Yaskawa INFORM job: miniTRJ2.JBI

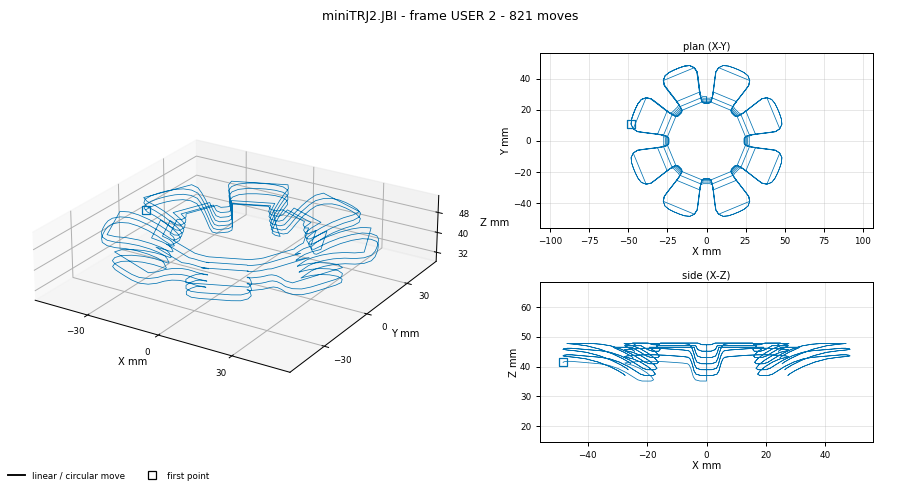
[picture p0: tool path of miniTRJ2.JBI in frame USER 2, 821 of 821 moves have a stored position in this frame; points joined in program order, loops and branches not executed]
/JOB
//NAME miniTRJ2
//POS
///NPOS 821,0,0,0,0,0
///USER 2
///TOOL 1
///POSTYPE USER
///RECTAN
///RCONF 1,0,0,0,0,0,0,0,0,0,0,0,0,0,0,0,0,0,0,0,0,0,0,0
C00000=-48.294,10.888,41.429,-176.7397,37.5709,0.0000
C00001=-47.960,14.116,41.642,-174.0482,36.6015,0.0000
C00002=-46.852,17.458,41.781,-171.5367,35.2544,0.0000
C00003=-45.474,20.785,41.781,148.5946,18.8544,0.0000
C00004=-43.894,23.932,41.642,148.9631,21.2691,0.0000
C00005=-41.848,26.450,41.429,149.6667,23.5333,0.0000
C00006=-38.982,27.526,41.216,150.5545,25.2242,0.0000
C00007=-35.890,26.937,40.953,151.2616,26.0383,0.0000
C00008=-32.968,24.818,40.447,151.5930,26.0678,0.0000
C00009=-29.853,22.391,39.399,151.8878,26.0592,0.0000
C00010=-27.005,20.165,37.988,152.1228,26.0805,0.0000
C00011=-24.775,18.500,36.587,152.2942,26.1489,0.0000
C00012=-23.134,17.826,35.561,152.5223,26.3895,0.0000
C00013=-21.719,18.610,35.152,153.0306,27.0004,0.0000
C00014=-20.847,19.522,35.134,152.8372,26.8332,0.0000
C00015=-20.193,20.193,35.146,151.5689,25.4617,0.0000
C00016=-19.522,20.846,35.134,150.3783,24.0388,0.0000
C00017=-18.610,21.719,35.152,150.2435,23.8342,0.0000
C00018=-17.826,23.134,35.561,150.7835,24.4140,0.0000
C00019=-18.500,24.775,36.587,150.9905,24.6675,0.0000
C00020=-20.165,27.005,37.988,151.0256,24.8329,0.0000
C00021=-22.391,29.853,39.399,150.9956,25.0433,0.0000
C00022=-24.818,32.968,40.447,150.9190,25.2991,0.0000
C00023=-26.937,35.890,40.953,150.8741,25.5955,0.0000
C00024=-27.526,38.982,41.216,151.5887,26.4057,0.0000
C00025=-26.450,41.848,41.429,153.2256,27.5826,0.0000
C00026=-23.932,43.894,41.642,155.5676,28.7163,0.0000
C00027=-20.785,45.474,41.781,158.1935,29.5466,0.0000
C00028=-17.458,46.852,41.781,144.4493,-6.9027,0.0000
C00029=-14.116,47.960,41.642,143.2501,-4.7750,0.0000
C00030=-10.888,48.294,41.429,142.3842,-2.5836,0.0000
C00031=-8.101,47.028,41.216,141.9857,-0.7523,0.0000
C00032=-6.331,44.425,40.953,141.9838,0.2816,0.0000
C00033=-5.763,40.861,40.447,142.1989,0.4896,0.0000
C00034=-5.276,36.942,39.399,142.4114,0.6478,0.0000
C00035=-4.837,33.354,37.988,142.5630,0.7963,0.0000
C00036=-4.437,30.601,36.587,142.6403,0.9460,0.0000
C00037=-3.753,28.963,35.561,142.6489,1.2616,0.0000
C00038=-2.199,28.517,35.152,142.6175,2.0220,0.0000
C00039=-0.937,28.545,35.134,142.5890,1.7848,0.0000
C00040=0.000,28.557,35.146,142.5588,-0.0019,0.0000
C00041=0.000,27.418,37.029,142.9317,-0.0022,0.0000
C00042=0.833,27.409,37.016,142.9601,-1.7182,0.0000
C00043=2.024,27.393,37.035,142.9884,-2.0087,0.0000
C00044=3.544,27.900,37.475,143.0157,-1.2641,0.0000
C00045=4.196,29.693,38.576,142.9980,-0.9669,0.0000
C00046=4.590,32.667,40.064,142.9030,-0.8249,0.0000
C00047=5.044,36.489,41.539,142.7233,-0.6720,0.0000
C00048=5.547,40.603,42.621,142.4757,-0.5065,0.0000
C00049=6.113,44.307,43.139,142.2242,-0.2970,0.0000
C00050=7.904,47.004,43.407,142.2019,0.7764,0.0000
C00051=10.737,48.321,43.623,142.6086,2.6858,0.0000
C00052=14.024,47.990,43.840,143.5265,4.9622,0.0000
C00053=17.428,46.864,43.981,144.8035,7.1518,0.0000
C00054=20.814,45.461,43.981,158.6858,-29.5002,0.0000
C00055=24.018,43.851,43.840,155.9451,-28.6807,0.0000
C00056=26.576,41.761,43.623,153.4943,-27.5200,0.0000
C00057=27.648,38.826,43.407,151.7943,-26.2899,0.0000
C00058=27.007,35.652,43.139,151.0729,-25.4348,0.0000
C00059=24.788,32.633,42.621,151.1478,-25.1145,0.0000
C00060=22.235,29.369,41.539,151.2491,-24.8312,0.0000
C00061=19.854,26.344,40.064,151.2998,-24.5999,0.0000
C00062=18.029,23.963,38.576,151.2850,-24.4296,0.0000
C00063=17.223,22.234,37.475,151.0981,-24.1854,0.0000
C00064=17.939,20.801,37.035,150.5715,-23.6167,0.0000
C00065=18.793,19.970,37.016,150.7430,-23.8628,0.0000
C00066=19.387,19.387,37.029,151.8889,-25.2262,0.0000
C00067=19.970,18.793,37.016,153.1137,-26.5489,0.0000
C00068=20.801,17.939,37.035,153.3424,-26.7551,0.0000
C00069=22.234,17.223,37.475,152.8415,-26.1602,0.0000
C00070=23.963,18.029,38.576,152.6183,-25.9402,0.0000
C00071=26.344,19.854,40.064,152.4370,-25.8893,0.0000
C00072=29.369,22.235,41.539,152.1749,-25.8826,0.0000
C00073=32.633,24.788,42.621,151.8451,-25.9079,0.0000
C00074=35.652,27.007,43.139,151.4812,-25.9004,0.0000
C00075=38.826,27.648,43.407,150.7258,-25.0713,0.0000
C00076=41.761,26.576,43.623,149.7917,-23.3150,0.0000
C00077=43.851,24.018,43.840,149.0753,-20.9529,0.0000
C00078=45.461,20.814,43.981,148.7289,-18.4429,0.0000
C00079=46.864,17.428,43.981,-171.2706,-34.8827,0.0000
C00080=47.990,14.024,43.840,-173.8375,-36.3149,0.0000
C00081=48.321,10.737,43.623,-176.6210,-37.3433,0.0000
C00082=47.004,7.904,43.407,-179.0175,-37.7940,0.0000
C00083=44.307,6.113,43.139,179.6243,-37.7752,0.0000
C00084=40.603,5.547,42.621,179.3613,-37.5226,0.0000
C00085=36.489,5.044,41.539,179.1555,-37.2737,0.0000
C00086=32.667,4.590,40.064,178.9658,-37.0926,0.0000
C00087=29.693,4.196,38.576,178.7894,-36.9959,0.0000
C00088=27.900,3.544,37.475,178.4177,-36.9738,0.0000
C00089=27.393,2.024,37.035,177.4851,-36.9851,0.0000
C00090=27.409,0.833,37.016,177.8479,-37.0204,0.0000
C00091=27.418,0.000,37.029,179.9973,-37.0683,0.0000
C00092=27.409,-0.832,37.016,-177.8467,-37.0204,0.0000
C00093=27.393,-2.024,37.035,-177.4859,-36.9851,0.0000
C00094=27.900,-3.544,37.475,-178.4183,-36.9738,0.0000
C00095=29.693,-4.196,38.576,-178.7900,-36.9959,0.0000
C00096=32.667,-4.590,40.064,-178.9664,-37.0925,0.0000
C00097=36.489,-5.044,41.539,-179.1560,-37.2737,0.0000
C00098=40.603,-5.547,42.621,-179.3619,-37.5226,0.0000
C00099=44.307,-6.113,43.139,-179.6249,-37.7752,0.0000
C00100=47.004,-7.904,43.407,179.0170,-37.7939,0.0000
C00101=48.321,-10.737,43.623,176.6207,-37.3433,0.0000
C00102=47.990,-14.024,43.840,173.8374,-36.3149,0.0000
C00103=46.864,-17.428,43.981,171.2706,-34.8827,0.0000
C00104=45.461,-20.814,43.981,-148.7290,-18.4429,0.0000
C00105=43.851,-24.018,43.840,-149.0753,-20.9529,0.0000
C00106=41.761,-26.576,43.623,-149.7918,-23.3152,0.0000
C00107=38.826,-27.648,43.407,-150.7260,-25.0716,0.0000
C00108=35.652,-27.007,43.139,-151.4815,-25.9008,0.0000
C00109=32.633,-24.788,42.621,-151.8454,-25.9083,0.0000
C00110=29.369,-22.235,41.539,-152.1752,-25.8829,0.0000
C00111=26.344,-19.854,40.064,-152.4373,-25.8897,0.0000
C00112=23.963,-18.029,38.576,-152.6186,-25.9406,0.0000
C00113=22.234,-17.223,37.475,-152.8418,-26.1606,0.0000
C00114=20.801,-17.939,37.035,-153.3429,-26.7556,0.0000
C00115=19.970,-18.793,37.016,-153.1131,-26.5482,0.0000
C00116=19.387,-19.387,37.029,-151.8919,-25.2296,0.0000
C00117=18.793,-19.970,37.016,-150.7424,-23.8621,0.0000
C00118=17.939,-20.801,37.035,-150.5720,-23.6172,0.0000
C00119=17.223,-22.234,37.475,-151.0984,-24.1858,0.0000
C00120=18.029,-23.963,38.576,-151.2853,-24.4300,0.0000
C00121=19.854,-26.344,40.064,-151.3001,-24.6002,0.0000
C00122=22.235,-29.369,41.539,-151.2494,-24.8316,0.0000
C00123=24.788,-32.633,42.621,-151.1482,-25.1149,0.0000
C00124=27.007,-35.652,43.139,-151.0733,-25.4352,0.0000
C00125=27.648,-38.826,43.407,-151.7946,-26.2902,0.0000
C00126=26.576,-41.761,43.623,-153.4945,-27.5201,0.0000
C00127=24.018,-43.851,43.840,-155.9452,-28.6808,0.0000
C00128=20.814,-45.461,43.981,-158.6857,-29.5002,0.0000
C00129=17.428,-46.864,43.981,-144.8035,7.1518,0.0000
C00130=14.024,-47.990,43.840,-143.5265,4.9622,0.0000
C00131=10.737,-48.321,43.623,-142.6086,2.6858,0.0000
C00132=7.904,-47.004,43.407,-142.2019,0.7764,0.0000
C00133=6.113,-44.307,43.139,-142.2242,-0.2970,0.0000
C00134=5.547,-40.603,42.621,-142.4757,-0.5065,0.0000
C00135=5.044,-36.489,41.539,-142.7233,-0.6720,0.0000
C00136=4.590,-32.667,40.064,-142.9030,-0.8249,0.0000
C00137=4.196,-29.693,38.576,-142.9980,-0.9669,0.0000
C00138=3.544,-27.900,37.475,-143.0157,-1.2641,0.0000
C00139=2.024,-27.393,37.035,-142.9884,-2.0087,0.0000
C00140=0.833,-27.409,37.016,-142.9601,-1.7182,0.0000
C00141=0.000,-27.418,37.029,-142.9317,-0.0022,0.0000
C00142=0.000,-27.418,37.029,-142.9317,-0.0022,0.0000
C00143=-0.832,-27.409,37.016,-142.9601,1.7191,0.0000
C00144=-2.024,-27.393,37.035,-142.9884,2.0080,0.0000
C00145=-3.544,-27.900,37.475,-143.0157,1.2636,0.0000
C00146=-4.196,-29.693,38.576,-142.9980,0.9664,0.0000
C00147=-4.590,-32.667,40.064,-142.9030,0.8245,0.0000
C00148=-5.044,-36.489,41.539,-142.7233,0.6716,0.0000
C00149=-5.547,-40.603,42.621,-142.4757,0.5061,0.0000
C00150=-6.113,-44.307,43.139,-142.2242,0.2965,0.0000
C00151=-7.904,-47.004,43.407,-142.2020,-0.7768,0.0000
C00152=-10.737,-48.321,43.623,-142.6086,-2.6860,0.0000
C00153=-14.024,-47.990,43.840,-143.5265,-4.9623,0.0000
C00154=-17.428,-46.864,43.981,-144.8035,-7.1518,0.0000
C00155=-20.814,-45.461,43.981,-158.6858,29.5002,0.0000
C00156=-24.018,-43.851,43.840,-155.9451,28.6807,0.0000
C00157=-26.576,-41.761,43.623,-153.4943,27.5200,0.0000
C00158=-27.648,-38.826,43.407,-151.7943,26.2899,0.0000
C00159=-27.007,-35.652,43.139,-151.0729,25.4348,0.0000
C00160=-24.788,-32.633,42.621,-151.1478,25.1145,0.0000
C00161=-22.235,-29.369,41.539,-151.2491,24.8312,0.0000
C00162=-19.854,-26.344,40.064,-151.2998,24.5999,0.0000
C00163=-18.029,-23.963,38.576,-151.2850,24.4296,0.0000
C00164=-17.223,-22.234,37.475,-151.0981,24.1854,0.0000
C00165=-17.939,-20.801,37.035,-150.5715,23.6167,0.0000
C00166=-18.793,-19.970,37.016,-150.7430,23.8628,0.0000
C00167=-19.387,-19.387,37.029,-151.8889,25.2262,0.0000
C00168=-19.970,-18.793,37.016,-153.1137,26.5489,0.0000
C00169=-20.801,-17.939,37.035,-153.3424,26.7551,0.0000
C00170=-22.234,-17.223,37.475,-152.8415,26.1602,0.0000
C00171=-23.963,-18.029,38.576,-152.6183,25.9402,0.0000
C00172=-26.344,-19.854,40.064,-152.4370,25.8893,0.0000
C00173=-29.369,-22.235,41.539,-152.1749,25.8826,0.0000
C00174=-32.633,-24.788,42.621,-151.8451,25.9079,0.0000
C00175=-35.652,-27.007,43.139,-151.4812,25.9004,0.0000
C00176=-38.826,-27.648,43.407,-150.7258,25.0713,0.0000
C00177=-41.761,-26.576,43.623,-149.7917,23.3150,0.0000
C00178=-43.851,-24.018,43.840,-149.0753,20.9529,0.0000
C00179=-45.461,-20.814,43.981,-148.7289,18.4429,0.0000
C00180=-46.864,-17.428,43.981,171.2706,34.8827,0.0000
C00181=-47.990,-14.024,43.840,173.8375,36.3149,0.0000
C00182=-48.321,-10.737,43.623,176.6210,37.3433,0.0000
C00183=-47.004,-7.904,43.407,179.0175,37.7940,0.0000
C00184=-44.307,-6.113,43.139,-179.6243,37.7752,0.0000
C00185=-40.603,-5.547,42.621,-179.3613,37.5226,0.0000
C00186=-36.489,-5.044,41.539,-179.1555,37.2737,0.0000
C00187=-32.667,-4.590,40.064,-178.9658,37.0926,0.0000
C00188=-29.693,-4.196,38.576,-178.7894,36.9959,0.0000
C00189=-27.900,-3.544,37.475,-178.4177,36.9738,0.0000
C00190=-27.393,-2.024,37.035,-177.4851,36.9851,0.0000
C00191=-27.409,-0.833,37.016,-177.8479,37.0204,0.0000
C00192=-27.418,0.000,37.029,-179.9973,37.0683,0.0000
C00193=-27.409,0.832,37.016,177.8467,37.0204,0.0000
C00194=-27.393,2.024,37.035,177.4859,36.9851,0.0000
C00195=-27.900,3.544,37.475,178.4183,36.9738,0.0000
C00196=-29.693,4.196,38.576,178.7900,36.9959,0.0000
C00197=-32.667,4.590,40.064,178.9664,37.0925,0.0000
C00198=-36.489,5.044,41.539,179.1560,37.2737,0.0000
C00199=-40.603,5.547,42.621,179.3619,37.5226,0.0000
C00200=-44.307,6.113,43.139,179.6249,37.7752,0.0000
C00201=-47.004,7.904,43.407,-179.0170,37.7939,0.0000
C00202=-48.321,10.737,43.623,-176.6207,37.3433,0.0000
C00203=-47.990,14.024,43.840,-173.8374,36.3149,0.0000
C00204=-46.864,17.428,43.981,-171.2706,34.8827,0.0000
C00205=-45.461,20.814,43.981,148.7290,18.4429,0.0000
C00206=-43.851,24.018,43.840,149.0753,20.9529,0.0000
C00207=-41.761,26.576,43.623,149.7918,23.3152,0.0000
C00208=-38.826,27.648,43.407,150.7260,25.0716,0.0000
C00209=-35.652,27.007,43.139,151.4815,25.9008,0.0000
C00210=-32.633,24.788,42.621,151.8454,25.9083,0.0000
C00211=-29.369,22.235,41.539,152.1752,25.8829,0.0000
C00212=-26.344,19.854,40.064,152.4373,25.8897,0.0000
C00213=-23.963,18.029,38.576,152.6186,25.9406,0.0000
C00214=-22.234,17.223,37.475,152.8418,26.1606,0.0000
C00215=-20.801,17.939,37.035,153.3429,26.7556,0.0000
C00216=-19.970,18.793,37.016,153.1131,26.5482,0.0000
C00217=-19.387,19.387,37.029,151.8919,25.2296,0.0000
C00218=-18.793,19.970,37.016,150.7424,23.8621,0.0000
C00219=-17.939,20.801,37.035,150.5720,23.6172,0.0000
C00220=-17.223,22.234,37.475,151.0984,24.1858,0.0000
C00221=-18.029,23.963,38.576,151.2853,24.4300,0.0000
C00222=-19.854,26.344,40.064,151.3001,24.6002,0.0000
C00223=-22.235,29.369,41.539,151.2494,24.8316,0.0000
C00224=-24.788,32.633,42.621,151.1482,25.1149,0.0000
C00225=-27.007,35.652,43.139,151.0733,25.4352,0.0000
C00226=-27.648,38.826,43.407,151.7946,26.2902,0.0000
C00227=-26.576,41.761,43.623,153.4945,27.5201,0.0000
C00228=-24.018,43.851,43.840,155.9452,28.6808,0.0000
C00229=-20.814,45.461,43.981,158.6857,29.5002,0.0000
C00230=-17.428,46.864,43.981,144.8035,-7.1518,0.0000
C00231=-14.024,47.990,43.840,143.5265,-4.9623,0.0000
C00232=-10.737,48.321,43.623,142.6086,-2.6860,0.0000
C00233=-7.904,47.004,43.407,142.2020,-0.7768,0.0000
C00234=-6.113,44.307,43.139,142.2242,0.2965,0.0000
C00235=-5.547,40.603,42.621,142.4757,0.5061,0.0000
C00236=-5.044,36.489,41.539,142.7233,0.6716,0.0000
C00237=-4.590,32.667,40.064,142.9030,0.8245,0.0000
C00238=-4.196,29.693,38.576,142.9980,0.9664,0.0000
C00239=-3.544,27.900,37.475,143.0157,1.2636,0.0000
C00240=-2.024,27.393,37.035,142.9884,2.0080,0.0000
C00241=-0.832,27.409,37.016,142.9601,1.7191,0.0000
C00242=0.000,27.418,37.029,142.9317,-0.0022,0.0000
C00243=0.000,26.383,38.970,143.3333,-0.0024,0.0000
C00244=0.738,26.377,38.956,143.3599,-1.6506,0.0000
C00245=1.865,26.371,38.977,143.3880,-1.9910,0.0000
C00246=3.355,26.945,39.448,143.4111,-1.2604,0.0000
C00247=3.987,28.902,40.618,143.3831,-0.9770,0.0000
C00248=4.387,32.102,42.180,143.2683,-0.8359,0.0000
C00249=4.868,36.145,43.705,143.0598,-0.6708,0.0000
C00250=5.395,40.422,44.808,142.7788,-0.4897,0.0000
C00251=5.967,44.227,45.333,142.4944,-0.2702,0.0000
C00252=7.777,46.989,45.603,142.4530,0.8448,0.0000
C00253=10.643,48.338,45.821,142.8730,2.8264,0.0000
C00254=13.968,48.009,46.039,143.8450,5.1732,0.0000
C00255=17.410,46.871,46.181,145.1966,7.4059,0.0000
C00256=20.832,45.453,46.181,159.2143,-29.4305,0.0000
C00257=24.070,43.824,46.039,156.3761,-28.6352,0.0000
C00258=26.655,41.706,45.821,153.8250,-27.4611,0.0000
C00259=27.727,38.725,45.603,152.0606,-26.1867,0.0000
C00260=27.054,35.493,45.333,151.3259,-25.2884,0.0000
C00261=24.768,32.397,44.808,151.4217,-24.9398,0.0000
C00262=22.116,29.001,43.705,151.5403,-24.6233,0.0000
C00263=19.598,25.801,42.180,151.6069,-24.3643,0.0000
C00264=17.618,23.256,40.618,151.6092,-24.1825,0.0000
C00265=16.680,21.426,39.448,151.4402,-23.9431,0.0000
C00266=17.329,19.966,38.977,150.9260,-23.3840,0.0000
C00267=18.130,19.173,38.956,151.1318,-23.6688,0.0000
C00268=18.656,18.656,38.970,152.2350,-24.9751,0.0000
C00269=19.173,18.130,38.956,153.4120,-26.2443,0.0000
C00270=19.966,17.329,38.977,153.6756,-26.4885,0.0000
C00271=21.426,16.680,39.448,153.1805,-25.9082,0.0000
C00272=23.256,17.618,40.618,152.9579,-25.7059,0.0000
C00273=25.801,19.598,42.180,152.7605,-25.6685,0.0000
C00274=29.001,22.116,43.705,152.4654,-25.6709,0.0000
C00275=32.397,24.768,44.808,152.0964,-25.7056,0.0000
C00276=35.493,27.054,45.333,151.6977,-25.7114,0.0000
C00277=38.725,27.727,45.603,150.8971,-24.8625,0.0000
C00278=41.706,26.655,45.821,149.9252,-23.0422,0.0000
C00279=43.824,24.070,46.039,149.2067,-20.5923,0.0000
C00280=45.453,20.832,46.181,148.8912,-18.0037,0.0000
C00281=46.871,17.410,46.181,-171.0047,-34.4718,0.0000
C00282=48.009,13.968,46.039,-173.6022,-35.9847,0.0000
C00283=48.338,10.643,45.821,-176.4566,-37.0743,0.0000
C00284=46.989,7.777,45.603,-178.9345,-37.5422,0.0000
C00285=44.227,5.967,45.333,179.6594,-37.5052,0.0000
C00286=40.422,5.395,44.808,179.3850,-37.2196,0.0000
C00287=36.145,4.868,43.705,179.1607,-36.9373,0.0000
C00288=32.102,4.387,42.180,178.9570,-36.7271,0.0000
C00289=28.902,3.987,40.618,178.7829,-36.6107,0.0000
C00290=26.945,3.355,39.448,178.4304,-36.5786,0.0000
C00291=26.371,1.865,38.977,177.5201,-36.5863,0.0000
C00292=26.377,0.738,38.956,177.9433,-36.6224,0.0000
C00293=26.383,0.000,38.970,179.9970,-36.6667,0.0000
C00294=26.377,-0.738,38.956,-177.9417,-36.6224,0.0000
C00295=26.371,-1.865,38.977,-177.5209,-36.5863,0.0000
C00296=26.945,-3.355,39.448,-178.4310,-36.5786,0.0000
C00297=28.902,-3.987,40.618,-178.7834,-36.6107,0.0000
C00298=32.102,-4.387,42.180,-178.9576,-36.7271,0.0000
C00299=36.145,-4.868,43.705,-179.1613,-36.9372,0.0000
C00300=40.422,-5.395,44.808,-179.3856,-37.2196,0.0000
C00301=44.227,-5.967,45.333,-179.6600,-37.5051,0.0000
C00302=46.989,-7.777,45.603,178.9341,-37.5421,0.0000
C00303=48.338,-10.643,45.821,176.4564,-37.0742,0.0000
C00304=48.009,-13.968,46.039,173.6022,-35.9847,0.0000
C00305=46.871,-17.410,46.181,171.0047,-34.4718,0.0000
C00306=45.453,-20.832,46.181,-148.8912,-18.0037,0.0000
C00307=43.824,-24.070,46.039,-149.2068,-20.5924,0.0000
C00308=41.706,-26.655,45.821,-149.9253,-23.0424,0.0000
C00309=38.725,-27.727,45.603,-150.8973,-24.8628,0.0000
C00310=35.493,-27.054,45.333,-151.6980,-25.7118,0.0000
C00311=32.397,-24.768,44.808,-152.0967,-25.7060,0.0000
C00312=29.001,-22.116,43.705,-152.4657,-25.6713,0.0000
C00313=25.801,-19.598,42.180,-152.7608,-25.6688,0.0000
C00314=23.256,-17.618,40.618,-152.9582,-25.7062,0.0000
C00315=21.426,-16.680,39.448,-153.1809,-25.9086,0.0000
C00316=19.966,-17.329,38.977,-153.6761,-26.4890,0.0000
C00317=19.173,-18.130,38.956,-153.4112,-26.2433,0.0000
C00318=18.656,-18.656,38.970,-152.2384,-24.9789,0.0000
C00319=18.130,-19.173,38.956,-151.1310,-23.6679,0.0000
C00320=17.329,-19.966,38.977,-150.9265,-23.3846,0.0000
C00321=16.680,-21.426,39.448,-151.4406,-23.9435,0.0000
C00322=17.618,-23.256,40.618,-151.6095,-24.1829,0.0000
C00323=19.598,-25.801,42.180,-151.6072,-24.3646,0.0000
C00324=22.116,-29.001,43.705,-151.5406,-24.6236,0.0000
C00325=24.768,-32.397,44.808,-151.4221,-24.9401,0.0000
C00326=27.054,-35.493,45.333,-151.3263,-25.2888,0.0000
C00327=27.727,-38.725,45.603,-152.0609,-26.1870,0.0000
C00328=26.655,-41.706,45.821,-153.8251,-27.4613,0.0000
C00329=24.070,-43.824,46.039,-156.3762,-28.6353,0.0000
C00330=20.832,-45.453,46.181,-159.2143,-29.4305,0.0000
C00331=17.410,-46.871,46.181,-145.1966,7.4059,0.0000
C00332=13.968,-48.009,46.039,-143.8450,5.1732,0.0000
C00333=10.643,-48.338,45.821,-142.8730,2.8264,0.0000
C00334=7.777,-46.989,45.603,-142.4530,0.8448,0.0000
C00335=5.967,-44.227,45.333,-142.4944,-0.2702,0.0000
C00336=5.395,-40.422,44.808,-142.7788,-0.4897,0.0000
C00337=4.868,-36.145,43.705,-143.0598,-0.6708,0.0000
C00338=4.387,-32.102,42.180,-143.2683,-0.8359,0.0000
C00339=3.987,-28.902,40.618,-143.3831,-0.9770,0.0000
C00340=3.355,-26.945,39.448,-143.4111,-1.2604,0.0000
C00341=1.865,-26.371,38.977,-143.3880,-1.9910,0.0000
C00342=0.738,-26.377,38.956,-143.3599,-1.6506,0.0000
C00343=0.000,-26.383,38.970,-143.3333,-0.0024,0.0000
C00344=0.000,-26.383,38.970,-143.3333,-0.0024,0.0000
C00345=-0.738,-26.377,38.956,-143.3599,1.6518,0.0000
C00346=-1.865,-26.371,38.977,-143.3880,1.9904,0.0000
C00347=-3.355,-26.945,39.448,-143.4111,1.2599,0.0000
C00348=-3.987,-28.902,40.618,-143.3831,0.9765,0.0000
C00349=-4.387,-32.102,42.180,-143.2684,0.8355,0.0000
C00350=-4.868,-36.145,43.705,-143.0598,0.6703,0.0000
C00351=-5.395,-40.422,44.808,-142.7788,0.4893,0.0000
C00352=-5.967,-44.227,45.333,-142.4944,0.2697,0.0000
C00353=-7.777,-46.989,45.603,-142.4531,-0.8452,0.0000
C00354=-10.643,-48.338,45.821,-142.8730,-2.8266,0.0000
C00355=-13.968,-48.009,46.039,-143.8450,-5.1732,0.0000
C00356=-17.410,-46.871,46.181,-145.1966,-7.4059,0.0000
C00357=-20.832,-45.453,46.181,-159.2143,29.4305,0.0000
C00358=-24.070,-43.824,46.039,-156.3761,28.6352,0.0000
C00359=-26.655,-41.706,45.821,-153.8250,27.4611,0.0000
C00360=-27.727,-38.725,45.603,-152.0606,26.1867,0.0000
C00361=-27.054,-35.493,45.333,-151.3259,25.2884,0.0000
C00362=-24.768,-32.397,44.808,-151.4217,24.9398,0.0000
C00363=-22.116,-29.001,43.705,-151.5403,24.6233,0.0000
C00364=-19.598,-25.801,42.180,-151.6069,24.3643,0.0000
C00365=-17.618,-23.256,40.618,-151.6092,24.1825,0.0000
C00366=-16.680,-21.426,39.448,-151.4402,23.9431,0.0000
C00367=-17.329,-19.966,38.977,-150.9260,23.3840,0.0000
C00368=-18.130,-19.173,38.956,-151.1318,23.6688,0.0000
C00369=-18.656,-18.656,38.970,-152.2350,24.9751,0.0000
C00370=-19.173,-18.130,38.956,-153.4120,26.2443,0.0000
C00371=-19.966,-17.329,38.977,-153.6756,26.4885,0.0000
C00372=-21.426,-16.680,39.448,-153.1805,25.9082,0.0000
C00373=-23.256,-17.618,40.618,-152.9579,25.7059,0.0000
C00374=-25.801,-19.598,42.180,-152.7605,25.6685,0.0000
C00375=-29.001,-22.116,43.705,-152.4654,25.6709,0.0000
C00376=-32.397,-24.768,44.808,-152.0964,25.7056,0.0000
C00377=-35.493,-27.054,45.333,-151.6977,25.7114,0.0000
C00378=-38.725,-27.727,45.603,-150.8971,24.8625,0.0000
C00379=-41.706,-26.655,45.821,-149.9252,23.0422,0.0000
C00380=-43.824,-24.070,46.039,-149.2067,20.5923,0.0000
C00381=-45.453,-20.832,46.181,-148.8912,18.0037,0.0000
C00382=-46.871,-17.410,46.181,171.0047,34.4718,0.0000
C00383=-48.009,-13.968,46.039,173.6022,35.9847,0.0000
C00384=-48.338,-10.643,45.821,176.4566,37.0743,0.0000
C00385=-46.989,-7.777,45.603,178.9345,37.5422,0.0000
C00386=-44.227,-5.967,45.333,-179.6594,37.5052,0.0000
C00387=-40.422,-5.395,44.808,-179.3850,37.2196,0.0000
C00388=-36.145,-4.868,43.705,-179.1607,36.9373,0.0000
C00389=-32.102,-4.387,42.180,-178.9570,36.7271,0.0000
C00390=-28.902,-3.987,40.618,-178.7829,36.6107,0.0000
C00391=-26.945,-3.355,39.448,-178.4304,36.5786,0.0000
C00392=-26.371,-1.865,38.977,-177.5201,36.5863,0.0000
C00393=-26.377,-0.738,38.956,-177.9433,36.6224,0.0000
C00394=-26.383,0.000,38.970,-179.9970,36.6667,0.0000
C00395=-26.377,0.738,38.956,177.9417,36.6224,0.0000
C00396=-26.371,1.865,38.977,177.5209,36.5863,0.0000
C00397=-26.945,3.355,39.448,178.4310,36.5786,0.0000
C00398=-28.902,3.987,40.618,178.7834,36.6107,0.0000
C00399=-32.102,4.387,42.180,178.9576,36.7271,0.0000
C00400=-36.145,4.868,43.705,179.1613,36.9372,0.0000
C00401=-40.422,5.395,44.808,179.3856,37.2196,0.0000
C00402=-44.227,5.967,45.333,179.6600,37.5051,0.0000
C00403=-46.989,7.777,45.603,-178.9341,37.5421,0.0000
C00404=-48.338,10.643,45.821,-176.4564,37.0742,0.0000
C00405=-48.009,13.968,46.039,-173.6022,35.9847,0.0000
C00406=-46.871,17.410,46.181,-171.0047,34.4718,0.0000
C00407=-45.453,20.832,46.181,148.8912,18.0037,0.0000
C00408=-43.824,24.070,46.039,149.2068,20.5924,0.0000
C00409=-41.706,26.655,45.821,149.9253,23.0424,0.0000
C00410=-38.725,27.727,45.603,150.8973,24.8628,0.0000
C00411=-35.493,27.054,45.333,151.6980,25.7118,0.0000
C00412=-32.397,24.768,44.808,152.0967,25.7060,0.0000
C00413=-29.001,22.116,43.705,152.4657,25.6713,0.0000
C00414=-25.801,19.598,42.180,152.7608,25.6688,0.0000
C00415=-23.256,17.618,40.618,152.9582,25.7062,0.0000
C00416=-21.426,16.680,39.448,153.1809,25.9086,0.0000
C00417=-19.966,17.329,38.977,153.6761,26.4890,0.0000
C00418=-19.173,18.130,38.956,153.4112,26.2433,0.0000
C00419=-18.656,18.656,38.970,152.2384,24.9789,0.0000
C00420=-18.130,19.173,38.956,151.1310,23.6679,0.0000
C00421=-17.329,19.966,38.977,150.9265,23.3846,0.0000
C00422=-16.680,21.426,39.448,151.4406,23.9435,0.0000
C00423=-17.618,23.256,40.618,151.6095,24.1829,0.0000
C00424=-19.598,25.801,42.180,151.6072,24.3646,0.0000
C00425=-22.116,29.001,43.705,151.5406,24.6236,0.0000
C00426=-24.768,32.397,44.808,151.4221,24.9401,0.0000
C00427=-27.054,35.493,45.333,151.3263,25.2888,0.0000
C00428=-27.727,38.725,45.603,152.0609,26.1870,0.0000
C00429=-26.655,41.706,45.821,153.8251,27.4613,0.0000
C00430=-24.070,43.824,46.039,156.3762,28.6353,0.0000
C00431=-20.832,45.453,46.181,159.2143,29.4305,0.0000
C00432=-17.410,46.871,46.181,145.1966,-7.4059,0.0000
C00433=-13.968,48.009,46.039,143.8450,-5.1732,0.0000
C00434=-10.643,48.338,45.821,142.8730,-2.8266,0.0000
C00435=-7.777,46.989,45.603,142.4531,-0.8452,0.0000
C00436=-5.967,44.227,45.333,142.4944,0.2697,0.0000
C00437=-5.395,40.422,44.808,142.7788,0.4893,0.0000
C00438=-4.868,36.145,43.705,143.0598,0.6703,0.0000
C00439=-4.387,32.102,42.180,143.2684,0.8355,0.0000
C00440=-3.987,28.902,40.618,143.3831,0.9765,0.0000
C00441=-3.355,26.945,39.448,143.4111,1.2599,0.0000
C00442=-1.865,26.371,38.977,143.3880,1.9904,0.0000
C00443=-0.738,26.377,38.956,143.3599,1.6518,0.0000
C00444=0.000,26.383,38.970,143.3333,-0.0024,0.0000
C00445=0.000,25.483,40.978,143.7606,-0.0027,0.0000
C00446=0.656,25.479,40.963,143.7854,-1.5834,0.0000
C00447=1.726,25.483,40.985,143.8134,-1.9683,0.0000
C00448=3.194,26.129,41.485,143.8318,-1.2486,0.0000
C00449=3.816,28.261,42.716,143.7915,-0.9729,0.0000
C00450=4.237,31.687,44.335,143.6546,-0.8247,0.0000
C00451=4.757,35.929,45.891,143.4171,-0.6383,0.0000
C00452=5.317,40.329,47.005,143.1061,-0.4321,0.0000
C00453=5.904,44.193,47.531,142.7941,-0.1927,0.0000
C00454=7.727,46.983,47.803,142.7410,0.9664,0.0000
C00455=27.758,38.686,47.803,152.3956,-26.1014,0.0000
C00456=27.074,35.424,47.531,151.6387,-25.1629,0.0000
C00457=24.758,32.277,47.005,151.7437,-24.7813,0.0000
C00458=22.041,28.769,45.891,151.8698,-24.4263,0.0000
C00459=19.410,25.402,44.335,151.9459,-24.1324,0.0000
C00460=17.285,22.682,42.716,151.9617,-23.9312,0.0000
C00461=16.217,20.734,41.485,151.8082,-23.6905,0.0000
C00462=16.798,19.240,40.985,151.3046,-23.1385,0.0000
C00463=17.553,18.480,40.963,151.5411,-23.4575,0.0000
C00464=18.019,18.019,40.978,152.6017,-24.7072,0.0000
C00465=18.480,17.553,40.963,153.7314,-25.9231,0.0000
C00466=19.240,16.798,40.985,154.0260,-26.2010,0.0000
C00467=20.735,16.217,41.485,153.5342,-25.6332,0.0000
C00468=22.682,17.285,42.716,153.3064,-25.4451,0.0000
C00469=25.402,19.410,44.335,153.0852,-25.4166,0.0000
C00470=28.769,22.041,45.891,152.7509,-25.4213,0.0000
C00471=32.277,24.758,47.005,152.3396,-25.4559,0.0000
C00472=35.424,27.074,47.531,151.9041,-25.4640,0.0000
C00473=38.686,27.758,47.803,151.0634,-24.5889,0.0000
C00474=46.983,7.727,47.803,-178.7859,-37.2528,0.0000
C00475=44.193,5.904,47.531,179.7580,-37.2056,0.0000
C00476=40.329,5.317,47.005,179.4597,-36.8927,0.0000
C00477=35.929,4.757,45.891,179.2051,-36.5803,0.0000
C00478=31.687,4.237,44.335,178.9761,-36.3410,0.0000
C00479=28.261,3.816,42.716,178.7942,-36.2024,0.0000
C00480=26.129,3.194,41.485,178.4534,-36.1582,0.0000
C00481=25.483,1.726,40.985,177.5617,-36.1619,0.0000
C00482=25.479,0.656,40.963,178.0377,-36.1986,0.0000
C00483=25.483,0.000,40.978,179.9967,-36.2394,0.0000
C00484=25.479,-0.655,40.963,-178.0358,-36.1986,0.0000
C00485=25.483,-1.727,40.985,-177.5626,-36.1619,0.0000
C00486=26.129,-3.194,41.485,-178.4540,-36.1582,0.0000
C00487=28.261,-3.816,42.716,-178.7948,-36.2024,0.0000
C00488=31.687,-4.237,44.335,-178.9767,-36.3410,0.0000
C00489=35.929,-4.757,45.891,-179.2056,-36.5803,0.0000
C00490=40.329,-5.317,47.005,-179.4603,-36.8926,0.0000
C00491=44.193,-5.904,47.531,-179.7586,-37.2056,0.0000
C00492=46.983,-7.727,47.803,178.7854,-37.2528,0.0000
C00493=38.686,-27.758,47.803,-151.0636,-24.5892,0.0000
C00494=35.424,-27.074,47.531,-151.9044,-25.4644,0.0000
C00495=32.277,-24.758,47.005,-152.3399,-25.4563,0.0000
C00496=28.769,-22.041,45.891,-152.7512,-25.4217,0.0000
C00497=25.402,-19.410,44.335,-153.0855,-25.4169,0.0000
C00498=22.682,-17.285,42.716,-153.3067,-25.4455,0.0000
C00499=20.734,-16.217,41.485,-153.5345,-25.6335,0.0000
C00500=19.240,-16.798,40.985,-154.0265,-26.2015,0.0000
C00501=18.480,-17.553,40.963,-153.7302,-25.9220,0.0000
C00502=18.019,-18.019,40.978,-152.6054,-24.7113,0.0000
C00503=17.553,-18.480,40.963,-151.5400,-23.4562,0.0000
C00504=16.798,-19.240,40.985,-151.3050,-23.1390,0.0000
C00505=16.217,-20.735,41.485,-151.8085,-23.6909,0.0000
C00506=17.285,-22.682,42.716,-151.9620,-23.9315,0.0000
C00507=19.410,-25.402,44.335,-151.9462,-24.1327,0.0000
C00508=22.041,-28.769,45.891,-151.8701,-24.4266,0.0000
C00509=24.758,-32.277,47.005,-151.7440,-24.7817,0.0000
C00510=27.074,-35.424,47.531,-151.6391,-25.1632,0.0000
C00511=27.758,-38.686,47.803,-152.3959,-26.1016,0.0000
C00512=7.727,-46.983,47.803,-142.7410,0.9664,0.0000
C00513=5.904,-44.193,47.531,-142.7941,-0.1927,0.0000
C00514=5.317,-40.329,47.005,-143.1061,-0.4321,0.0000
C00515=4.757,-35.929,45.891,-143.4171,-0.6383,0.0000
C00516=4.237,-31.687,44.335,-143.6546,-0.8247,0.0000
C00517=3.816,-28.261,42.716,-143.7915,-0.9729,0.0000
C00518=3.194,-26.129,41.485,-143.8318,-1.2486,0.0000
C00519=1.726,-25.483,40.985,-143.8134,-1.9683,0.0000
C00520=0.656,-25.479,40.963,-143.7854,-1.5834,0.0000
C00521=0.000,-25.483,40.978,-143.7606,-0.0027,0.0000
C00522=0.000,-25.483,40.978,-143.7606,-0.0027,0.0000
C00523=-0.655,-25.479,40.963,-143.7854,1.5850,0.0000
C00524=-1.727,-25.483,40.985,-143.8134,1.9677,0.0000
C00525=-3.194,-26.129,41.485,-143.8318,1.2481,0.0000
C00526=-3.816,-28.261,42.716,-143.7915,0.9725,0.0000
C00527=-4.237,-31.687,44.335,-143.6547,0.8243,0.0000
C00528=-4.757,-35.929,45.891,-143.4171,0.6379,0.0000
C00529=-5.317,-40.329,47.005,-143.1061,0.4317,0.0000
C00530=-5.904,-44.193,47.531,-142.7942,0.1923,0.0000
C00531=-7.727,-46.983,47.803,-142.7410,-0.9667,0.0000
C00532=-27.758,-38.686,47.803,-152.3956,26.1014,0.0000
C00533=-27.074,-35.424,47.531,-151.6387,25.1629,0.0000
C00534=-24.758,-32.277,47.005,-151.7437,24.7813,0.0000
C00535=-22.041,-28.769,45.891,-151.8698,24.4263,0.0000
C00536=-19.410,-25.402,44.335,-151.9459,24.1324,0.0000
C00537=-17.285,-22.682,42.716,-151.9617,23.9312,0.0000
C00538=-16.217,-20.734,41.485,-151.8082,23.6905,0.0000
C00539=-16.798,-19.240,40.985,-151.3046,23.1385,0.0000
C00540=-17.553,-18.480,40.963,-151.5411,23.4575,0.0000
C00541=-18.019,-18.019,40.978,-152.6017,24.7072,0.0000
C00542=-18.480,-17.553,40.963,-153.7314,25.9231,0.0000
C00543=-19.240,-16.798,40.985,-154.0260,26.2010,0.0000
C00544=-20.735,-16.217,41.485,-153.5342,25.6332,0.0000
C00545=-22.682,-17.285,42.716,-153.3064,25.4451,0.0000
C00546=-25.402,-19.410,44.335,-153.0852,25.4166,0.0000
C00547=-28.769,-22.041,45.891,-152.7509,25.4213,0.0000
C00548=-32.277,-24.758,47.005,-152.3396,25.4559,0.0000
C00549=-35.424,-27.074,47.531,-151.9041,25.4640,0.0000
C00550=-38.686,-27.758,47.803,-151.0634,24.5889,0.0000
C00551=-46.983,-7.727,47.803,178.7859,37.2528,0.0000
C00552=-44.193,-5.904,47.531,-179.7580,37.2056,0.0000
C00553=-40.329,-5.317,47.005,-179.4597,36.8927,0.0000
C00554=-35.929,-4.757,45.891,-179.2051,36.5803,0.0000
C00555=-31.687,-4.237,44.335,-178.9761,36.3410,0.0000
C00556=-28.261,-3.816,42.716,-178.7942,36.2024,0.0000
C00557=-26.129,-3.194,41.485,-178.4534,36.1582,0.0000
C00558=-25.483,-1.726,40.985,-177.5617,36.1619,0.0000
C00559=-25.479,-0.656,40.963,-178.0377,36.1986,0.0000
C00560=-25.483,0.000,40.978,-179.9967,36.2394,0.0000
C00561=-25.479,0.655,40.963,178.0358,36.1986,0.0000
C00562=-25.483,1.727,40.985,177.5626,36.1619,0.0000
C00563=-26.129,3.194,41.485,178.4540,36.1582,0.0000
C00564=-28.261,3.816,42.716,178.7948,36.2024,0.0000
C00565=-31.687,4.237,44.335,178.9767,36.3410,0.0000
C00566=-35.929,4.757,45.891,179.2056,36.5803,0.0000
C00567=-40.329,5.317,47.005,179.4603,36.8926,0.0000
C00568=-44.193,5.904,47.531,179.7586,37.2056,0.0000
C00569=-46.983,7.727,47.803,-178.7854,37.2528,0.0000
C00570=-38.686,27.758,47.803,151.0636,24.5892,0.0000
C00571=-35.424,27.074,47.531,151.9044,25.4644,0.0000
C00572=-32.277,24.758,47.005,152.3399,25.4563,0.0000
C00573=-28.769,22.041,45.891,152.7512,25.4217,0.0000
C00574=-25.402,19.410,44.335,153.0855,25.4169,0.0000
C00575=-22.682,17.285,42.716,153.3067,25.4455,0.0000
C00576=-20.734,16.217,41.485,153.5345,25.6335,0.0000
C00577=-19.240,16.798,40.985,154.0265,26.2015,0.0000
C00578=-18.480,17.553,40.963,153.7302,25.9220,0.0000
C00579=-18.019,18.019,40.978,152.6054,24.7113,0.0000
C00580=-17.553,18.480,40.963,151.5400,23.4562,0.0000
C00581=-16.798,19.240,40.985,151.3050,23.1390,0.0000
C00582=-16.217,20.735,41.485,151.8085,23.6909,0.0000
C00583=-17.285,22.682,42.716,151.9620,23.9315,0.0000
C00584=-19.410,25.402,44.335,151.9462,24.1327,0.0000
C00585=-22.041,28.769,45.891,151.8701,24.4266,0.0000
C00586=-24.758,32.277,47.005,151.7440,24.7817,0.0000
C00587=-27.074,35.424,47.531,151.6391,25.1632,0.0000
C00588=-27.758,38.686,47.803,152.3959,26.1016,0.0000
C00589=-7.727,46.983,47.803,142.7410,-0.9667,0.0000
C00590=-5.904,44.193,47.531,142.7942,0.1923,0.0000
C00591=-5.317,40.329,47.005,143.1061,0.4317,0.0000
C00592=-4.757,35.929,45.891,143.4171,0.6379,0.0000
C00593=-4.237,31.687,44.335,143.6547,0.8243,0.0000
C00594=-3.816,28.261,42.716,143.7915,0.9725,0.0000
C00595=-3.194,26.129,41.485,143.8318,1.2481,0.0000
C00596=-1.727,25.483,40.985,143.8134,1.9677,0.0000
C00597=-0.655,25.479,40.963,143.7854,1.5850,0.0000
C00598=0.000,25.483,40.978,143.7606,-0.0027,0.0000
C00599=0.000,24.757,43.054,144.2085,-0.0028,0.0000
C00600=0.589,24.754,43.039,144.2318,-1.5200,0.0000
C00601=1.615,24.766,43.062,144.2597,-1.9391,0.0000
C00602=3.068,25.489,43.586,144.2726,-1.2260,0.0000
C00603=3.695,27.804,44.865,144.2172,-0.9506,0.0000
C00604=4.151,31.448,46.521,144.0556,-0.7859,0.0000
C00605=19.301,25.172,46.521,152.3151,-23.9121,0.0000
C00606=17.048,22.273,44.865,152.3400,-23.6825,0.0000
C00607=15.854,20.193,43.586,152.1991,-23.4330,0.0000
C00608=16.370,18.654,43.062,151.7039,-22.8840,0.0000
C00609=17.087,17.920,43.039,151.9643,-23.2290,0.0000
C00610=17.506,17.506,43.054,152.9846,-24.4253,0.0000
C00611=17.920,17.087,43.039,154.0695,-25.5909,0.0000
C00612=18.654,16.370,43.062,154.3879,-25.8943,0.0000
C00613=20.193,15.854,43.586,153.8957,-25.3362,0.0000
C00614=22.273,17.048,44.865,153.6552,-25.1586,0.0000
C00615=25.172,19.301,46.521,153.4019,-25.1333,0.0000
C00616=31.448,4.151,46.521,179.0293,-35.9405,0.0000
C00617=27.804,3.695,44.865,178.8283,-35.7772,0.0000
C00618=25.489,3.068,43.586,178.4899,-35.7179,0.0000
C00619=24.766,1.615,43.062,177.6115,-35.7167,0.0000
C00620=24.754,0.589,43.039,178.1269,-35.7537,0.0000
C00621=24.757,0.000,43.054,179.9965,-35.7915,0.0000
C00622=24.754,-0.589,43.039,-178.1246,-35.7536,0.0000
C00623=24.766,-1.615,43.062,-177.6123,-35.7167,0.0000
C00624=25.489,-3.068,43.586,-178.4905,-35.7179,0.0000
C00625=27.804,-3.695,44.865,-178.8288,-35.7772,0.0000
C00626=31.448,-4.151,46.521,-179.0299,-35.9405,0.0000
C00627=25.172,-19.301,46.521,-153.4022,-25.1336,0.0000
C00628=22.273,-17.048,44.865,-153.6555,-25.1589,0.0000
C00629=20.193,-15.854,43.586,-153.8961,-25.3366,0.0000
C00630=18.654,-16.370,43.062,-154.3884,-25.8948,0.0000
C00631=17.920,-17.087,43.039,-154.0682,-25.5895,0.0000
C00632=17.506,-17.506,43.054,-152.9885,-24.4298,0.0000
C00633=17.087,-17.920,43.039,-151.9631,-23.2275,0.0000
C00634=16.370,-18.654,43.062,-151.7043,-22.8846,0.0000
C00635=15.854,-20.193,43.586,-152.1994,-23.4334,0.0000
C00636=17.048,-22.273,44.865,-152.3403,-23.6828,0.0000
C00637=19.301,-25.172,46.521,-152.3154,-23.9124,0.0000
C00638=4.151,-31.448,46.521,-144.0556,-0.7859,0.0000
C00639=3.695,-27.804,44.865,-144.2172,-0.9506,0.0000
C00640=3.068,-25.489,43.586,-144.2726,-1.2260,0.0000
C00641=1.615,-24.766,43.062,-144.2597,-1.9391,0.0000
C00642=0.589,-24.754,43.039,-144.2318,-1.5200,0.0000
C00643=0.000,-24.757,43.054,-144.2085,-0.0028,0.0000
C00644=0.000,-24.757,43.054,-144.2085,-0.0028,0.0000
C00645=-0.589,-24.754,43.039,-144.2319,1.5218,0.0000
C00646=-1.615,-24.766,43.062,-144.2597,1.9384,0.0000
C00647=-3.068,-25.489,43.586,-144.2726,1.2255,0.0000
C00648=-3.695,-27.804,44.865,-144.2172,0.9502,0.0000
C00649=-4.151,-31.448,46.521,-144.0556,0.7854,0.0000
C00650=-19.301,-25.172,46.521,-152.3151,23.9121,0.0000
C00651=-17.048,-22.273,44.865,-152.3400,23.6825,0.0000
C00652=-15.854,-20.193,43.586,-152.1991,23.4330,0.0000
C00653=-16.370,-18.654,43.062,-151.7039,22.8840,0.0000
C00654=-17.087,-17.920,43.039,-151.9643,23.2290,0.0000
C00655=-17.506,-17.506,43.054,-152.9846,24.4253,0.0000
C00656=-17.920,-17.087,43.039,-154.0695,25.5909,0.0000
C00657=-18.654,-16.370,43.062,-154.3879,25.8943,0.0000
C00658=-20.193,-15.854,43.586,-153.8957,25.3362,0.0000
C00659=-22.273,-17.048,44.865,-153.6552,25.1586,0.0000
C00660=-25.172,-19.301,46.521,-153.4019,25.1333,0.0000
C00661=-31.448,-4.151,46.521,-179.0293,35.9405,0.0000
C00662=-27.804,-3.695,44.865,-178.8283,35.7772,0.0000
C00663=-25.489,-3.068,43.586,-178.4899,35.7179,0.0000
C00664=-24.766,-1.615,43.062,-177.6115,35.7167,0.0000
C00665=-24.754,-0.589,43.039,-178.1269,35.7537,0.0000
C00666=-24.757,0.000,43.054,-179.9965,35.7915,0.0000
C00667=-24.754,0.589,43.039,178.1246,35.7536,0.0000
C00668=-24.766,1.615,43.062,177.6123,35.7167,0.0000
C00669=-25.489,3.068,43.586,178.4905,35.7179,0.0000
C00670=-27.804,3.695,44.865,178.8288,35.7772,0.0000
C00671=-31.448,4.151,46.521,179.0299,35.9405,0.0000
C00672=-25.172,19.301,46.521,153.4022,25.1336,0.0000
C00673=-22.273,17.048,44.865,153.6555,25.1589,0.0000
C00674=-20.193,15.854,43.586,153.8961,25.3366,0.0000
C00675=-18.654,16.370,43.062,154.3884,25.8948,0.0000
C00676=-17.920,17.087,43.039,154.0682,25.5895,0.0000
C00677=-17.506,17.506,43.054,152.9885,24.4298,0.0000
C00678=-17.087,17.920,43.039,151.9631,23.2275,0.0000
C00679=-16.370,18.654,43.062,151.7043,22.8846,0.0000
C00680=-15.854,20.193,43.586,152.1994,23.4334,0.0000
C00681=-17.048,22.273,44.865,152.3403,23.6828,0.0000
C00682=-19.301,25.172,46.521,152.3154,23.9124,0.0000
C00683=-4.151,31.448,46.521,144.0556,0.7854,0.0000
C00684=-3.695,27.804,44.865,144.2172,0.9502,0.0000
C00685=-3.068,25.489,43.586,144.2726,1.2255,0.0000
C00686=-1.615,24.766,43.062,144.2597,1.9384,0.0000
C00687=-0.589,24.754,43.039,144.2319,1.5218,0.0000
C00688=0.000,24.757,43.054,144.2085,-0.0028,0.0000
C00689=0.000,24.250,45.195,144.6693,-0.0030,0.0000
C00690=0.543,24.247,45.179,144.6915,-1.4646,0.0000
C00691=1.537,24.267,45.203,144.7189,-1.9015,0.0000
C00692=2.986,25.071,45.744,144.7252,-1.1893,0.0000
C00693=3.633,27.569,47.051,144.6512,-0.9055,0.0000
C00694=16.925,22.063,47.051,152.7394,-23.4452,0.0000
C00695=15.616,19.839,45.744,152.6079,-23.1780,0.0000
C00696=16.072,18.246,45.203,152.1182,-22.6269,0.0000
C00697=16.761,17.529,45.179,152.3917,-22.9847,0.0000
C00698=17.148,17.148,45.195,153.3766,-24.1345,0.0000
C00699=17.529,16.762,45.179,154.4228,-25.2557,0.0000
C00700=18.246,16.072,45.203,154.7533,-25.5721,0.0000
C00701=19.839,15.616,45.744,154.2558,-25.0201,0.0000
C00702=22.063,16.925,47.051,153.9937,-24.8483,0.0000
C00703=27.569,3.633,47.051,178.8898,-35.3437,0.0000
C00704=25.071,2.986,45.744,178.5433,-35.2661,0.0000
C00705=24.267,1.537,45.203,177.6710,-35.2587,0.0000
C00706=24.247,0.543,45.179,178.2054,-35.2953,0.0000
C00707=24.250,0.000,45.195,179.9964,-35.3307,0.0000
C00708=24.247,-0.542,45.179,-178.2028,-35.2952,0.0000
C00709=24.267,-1.537,45.203,-177.6719,-35.2588,0.0000
C00710=25.071,-2.986,45.744,-178.5439,-35.2661,0.0000
C00711=27.569,-3.633,47.051,-178.8904,-35.3437,0.0000
C00712=22.063,-16.925,47.051,-153.9940,-24.8486,0.0000
C00713=19.839,-15.616,45.744,-154.2561,-25.0205,0.0000
C00714=18.246,-16.072,45.203,-154.7538,-25.5726,0.0000
C00715=17.529,-16.761,45.179,-154.4213,-25.2541,0.0000
C00716=17.148,-17.148,45.195,-153.3807,-24.1391,0.0000
C00717=16.762,-17.529,45.179,-152.3903,-22.9831,0.0000
C00718=16.072,-18.246,45.203,-152.1186,-22.6274,0.0000
C00719=15.616,-19.839,45.744,-152.6083,-23.1783,0.0000
C00720=16.925,-22.063,47.051,-152.7397,-23.4456,0.0000
C00721=3.633,-27.569,47.051,-144.6512,-0.9055,0.0000
C00722=2.986,-25.071,45.744,-144.7252,-1.1893,0.0000
C00723=1.537,-24.267,45.203,-144.7189,-1.9015,0.0000
C00724=0.543,-24.247,45.179,-144.6915,-1.4646,0.0000
C00725=0.000,-24.250,45.195,-144.6693,-0.0030,0.0000
C00726=0.000,-24.250,45.195,-144.6693,-0.0030,0.0000
C00727=-0.542,-24.247,45.179,-144.6915,1.4667,0.0000
C00728=-1.537,-24.267,45.203,-144.7189,1.9009,0.0000
C00729=-2.986,-25.071,45.744,-144.7252,1.1889,0.0000
C00730=-3.633,-27.569,47.051,-144.6512,0.9051,0.0000
C00731=-16.925,-22.063,47.051,-152.7394,23.4452,0.0000
C00732=-15.616,-19.839,45.744,-152.6079,23.1780,0.0000
C00733=-16.072,-18.246,45.203,-152.1182,22.6269,0.0000
C00734=-16.761,-17.529,45.179,-152.3917,22.9847,0.0000
C00735=-17.148,-17.148,45.195,-153.3766,24.1345,0.0000
C00736=-17.529,-16.762,45.179,-154.4228,25.2557,0.0000
C00737=-18.246,-16.072,45.203,-154.7533,25.5721,0.0000
C00738=-19.839,-15.616,45.744,-154.2558,25.0201,0.0000
C00739=-22.063,-16.925,47.051,-153.9937,24.8483,0.0000
C00740=-27.569,-3.633,47.051,-178.8898,35.3437,0.0000
C00741=-25.071,-2.986,45.744,-178.5433,35.2661,0.0000
C00742=-24.267,-1.537,45.203,-177.6710,35.2587,0.0000
C00743=-24.247,-0.543,45.179,-178.2054,35.2953,0.0000
C00744=-24.250,0.000,45.195,-179.9964,35.3307,0.0000
C00745=-24.247,0.542,45.179,178.2028,35.2952,0.0000
C00746=-24.267,1.537,45.203,177.6719,35.2588,0.0000
C00747=-25.071,2.986,45.744,178.5439,35.2661,0.0000
C00748=-27.569,3.633,47.051,178.8904,35.3437,0.0000
C00749=-22.063,16.925,47.051,153.9940,24.8486,0.0000
C00750=-19.839,15.616,45.744,154.2561,25.0205,0.0000
C00751=-18.246,16.072,45.203,154.7538,25.5726,0.0000
C00752=-17.529,16.761,45.179,154.4213,25.2541,0.0000
C00753=-17.148,17.148,45.195,153.3807,24.1391,0.0000
C00754=-16.762,17.529,45.179,152.3903,22.9831,0.0000
C00755=-16.072,18.246,45.203,152.1186,22.6274,0.0000
C00756=-15.616,19.839,45.744,152.6083,23.1783,0.0000
C00757=-16.925,22.063,47.051,152.7397,23.4456,0.0000
C00758=-3.633,27.569,47.051,144.6512,0.9051,0.0000
C00759=-2.986,25.071,45.744,144.7252,1.1889,0.0000
C00760=-1.537,24.267,45.203,144.7189,1.9009,0.0000
C00761=-0.542,24.247,45.179,144.6915,1.4667,0.0000
C00762=0.000,24.250,45.195,144.6693,-0.0030,0.0000
C00763=0.000,24.012,47.382,145.1309,-0.0030,0.0000
C00764=0.521,24.008,47.366,145.1526,-1.4225,0.0000
C00765=1.501,24.033,47.390,145.1793,-1.8542,0.0000
C00766=2.955,24.917,47.939,145.1775,-1.1357,0.0000
C00767=15.529,19.709,47.939,153.0267,-22.9351,0.0000
C00768=15.933,18.055,47.390,152.5384,-22.3755,0.0000
C00769=16.608,17.344,47.366,152.8097,-22.7280,0.0000
C00770=16.979,16.979,47.382,153.7676,-23.8422,0.0000
C00771=17.344,16.608,47.366,154.7847,-24.9288,0.0000
C00772=18.055,15.933,47.390,155.1107,-25.2409,0.0000
C00773=19.709,15.529,47.939,154.6019,-24.6903,0.0000
C00774=24.917,2.955,47.939,178.6166,-34.8146,0.0000
C00775=24.033,1.501,47.390,177.7417,-34.7998,0.0000
C00776=24.008,0.521,47.366,178.2668,-34.8351,0.0000
C00777=24.012,0.000,47.382,179.9963,-34.8691,0.0000
C00778=24.008,-0.521,47.366,-178.2642,-34.8350,0.0000
C00779=24.033,-1.501,47.390,-177.7425,-34.7999,0.0000
C00780=24.917,-2.955,47.939,-178.6172,-34.8146,0.0000
C00781=19.709,-15.529,47.939,-154.6022,-24.6907,0.0000
C00782=18.055,-15.933,47.390,-155.1112,-25.2414,0.0000
C00783=17.344,-16.608,47.366,-154.7831,-24.9271,0.0000
C00784=16.979,-16.979,47.382,-153.7718,-23.8469,0.0000
C00785=16.608,-17.344,47.366,-152.8082,-22.7263,0.0000
C00786=15.933,-18.055,47.390,-152.5388,-22.3760,0.0000
C00787=15.529,-19.709,47.939,-153.0270,-22.9355,0.0000
C00788=2.955,-24.917,47.939,-145.1775,-1.1357,0.0000
C00789=1.501,-24.033,47.390,-145.1793,-1.8542,0.0000
C00790=0.521,-24.008,47.366,-145.1526,-1.4225,0.0000
C00791=0.000,-24.012,47.382,-145.1309,-0.0030,0.0000
C00792=0.000,-24.012,47.382,-145.1309,-0.0030,0.0000
C00793=-0.521,-24.008,47.366,-145.1526,1.4247,0.0000
C00794=-1.501,-24.033,47.390,-145.1793,1.8536,0.0000
C00795=-2.955,-24.917,47.939,-145.1775,1.1352,0.0000
C00796=-15.529,-19.709,47.939,-153.0267,22.9351,0.0000
C00797=-15.933,-18.055,47.390,-152.5384,22.3755,0.0000
C00798=-16.608,-17.344,47.366,-152.8097,22.7280,0.0000
C00799=-16.979,-16.979,47.382,-153.7676,23.8422,0.0000
C00800=-17.344,-16.608,47.366,-154.7847,24.9288,0.0000
C00801=-18.055,-15.933,47.390,-155.1107,25.2409,0.0000
C00802=-19.709,-15.529,47.939,-154.6019,24.6903,0.0000
C00803=-24.917,-2.955,47.939,-178.6166,34.8146,0.0000
C00804=-24.033,-1.501,47.390,-177.7417,34.7998,0.0000
C00805=-24.008,-0.521,47.366,-178.2668,34.8351,0.0000
C00806=-24.012,0.000,47.382,-179.9963,34.8691,0.0000
C00807=-24.008,0.521,47.366,178.2642,34.8350,0.0000
C00808=-24.033,1.501,47.390,177.7425,34.7999,0.0000
C00809=-24.917,2.955,47.939,178.6172,34.8146,0.0000
C00810=-19.709,15.529,47.939,154.6022,24.6907,0.0000
C00811=-18.055,15.933,47.390,155.1112,25.2414,0.0000
C00812=-17.344,16.608,47.366,154.7831,24.9271,0.0000
C00813=-16.979,16.979,47.382,153.7718,23.8469,0.0000
C00814=-16.608,17.344,47.366,152.8082,22.7263,0.0000
C00815=-15.933,18.055,47.390,152.5388,22.3760,0.0000
C00816=-15.529,19.709,47.939,153.0270,22.9355,0.0000
C00817=-2.955,24.917,47.939,145.1775,1.1352,0.0000
C00818=-1.501,24.033,47.390,145.1793,1.8536,0.0000
C00819=-0.521,24.008,47.366,145.1526,1.4247,0.0000
C00820=0.000,24.012,47.382,145.1309,-0.0030,0.0000
//INST
///DATE 2021/02/10 13:51
///COMM
///ATTR SC,RW,RJ
////FRAME USER 2
///GROUP1 RB1
NOP
MOVL C00000
MOVL C00001
MOVL C00002
MOVL C00003
MOVL C00004
MOVL C00005
MOVL C00006
MOVL C00007
MOVL C00008
MOVL C00009
MOVL C00010
MOVL C00011
MOVL C00012
MOVL C00013
MOVL C00014
MOVL C00015
MOVL C00016
MOVL C00017
MOVL C00018
MOVL C00019
MOVL C00020
MOVL C00021
MOVL C00022
MOVL C00023
MOVL C00024
MOVL C00025
MOVL C00026
MOVL C00027
MOVL C00028
MOVL C00029
MOVL C00030
MOVL C00031
MOVL C00032
MOVL C00033
MOVL C00034
MOVL C00035
MOVL C00036
MOVL C00037
MOVL C00038
MOVL C00039
MOVL C00040
MOVL C00041
MOVL C00042
MOVL C00043
MOVL C00044
MOVL C00045
MOVL C00046
MOVL C00047
MOVL C00048
MOVL C00049
MOVL C00050
MOVL C00051
MOVL C00052
MOVL C00053
MOVL C00054
MOVL C00055
MOVL C00056
MOVL C00057
MOVL C00058
MOVL C00059
MOVL C00060
MOVL C00061
MOVL C00062
MOVL C00063
MOVL C00064
MOVL C00065
MOVL C00066
MOVL C00067
MOVL C00068
MOVL C00069
MOVL C00070
MOVL C00071
MOVL C00072
MOVL C00073
MOVL C00074
MOVL C00075
MOVL C00076
MOVL C00077
MOVL C00078
MOVL C00079
MOVL C00080
MOVL C00081
MOVL C00082
MOVL C00083
MOVL C00084
MOVL C00085
MOVL C00086
MOVL C00087
MOVL C00088
MOVL C00089
MOVL C00090
MOVL C00091
MOVL C00092
MOVL C00093
MOVL C00094
MOVL C00095
MOVL C00096
MOVL C00097
MOVL C00098
MOVL C00099
MOVL C00100
MOVL C00101
MOVL C00102
MOVL C00103
MOVL C00104
MOVL C00105
MOVL C00106
MOVL C00107
MOVL C00108
MOVL C00109
MOVL C00110
MOVL C00111
MOVL C00112
MOVL C00113
MOVL C00114
MOVL C00115
MOVL C00116
MOVL C00117
MOVL C00118
MOVL C00119
MOVL C00120
MOVL C00121
MOVL C00122
MOVL C00123
MOVL C00124
MOVL C00125
MOVL C00126
MOVL C00127
MOVL C00128
MOVL C00129
MOVL C00130
MOVL C00131
MOVL C00132
MOVL C00133
MOVL C00134
MOVL C00135
MOVL C00136
MOVL C00137
MOVL C00138
MOVL C00139
MOVL C00140
MOVL C00141
MOVL C00142
MOVL C00143
MOVL C00144
MOVL C00145
MOVL C00146
MOVL C00147
MOVL C00148
MOVL C00149
MOVL C00150
MOVL C00151
MOVL C00152
MOVL C00153
MOVL C00154
MOVL C00155
MOVL C00156
MOVL C00157
MOVL C00158
MOVL C00159
MOVL C00160
MOVL C00161
MOVL C00162
MOVL C00163
MOVL C00164
MOVL C00165
MOVL C00166
MOVL C00167
MOVL C00168
MOVL C00169
MOVL C00170
MOVL C00171
MOVL C00172
MOVL C00173
MOVL C00174
MOVL C00175
MOVL C00176
MOVL C00177
MOVL C00178
MOVL C00179
MOVL C00180
MOVL C00181
MOVL C00182
MOVL C00183
MOVL C00184
MOVL C00185
MOVL C00186
MOVL C00187
MOVL C00188
MOVL C00189
MOVL C00190
MOVL C00191
MOVL C00192
MOVL C00193
MOVL C00194
MOVL C00195
MOVL C00196
MOVL C00197
MOVL C00198
MOVL C00199
MOVL C00200
MOVL C00201
MOVL C00202
MOVL C00203
MOVL C00204
MOVL C00205
MOVL C00206
MOVL C00207
MOVL C00208
MOVL C00209
MOVL C00210
MOVL C00211
MOVL C00212
MOVL C00213
MOVL C00214
MOVL C00215
MOVL C00216
MOVL C00217
MOVL C00218
MOVL C00219
MOVL C00220
MOVL C00221
MOVL C00222
MOVL C00223
MOVL C00224
MOVL C00225
MOVL C00226
MOVL C00227
MOVL C00228
MOVL C00229
MOVL C00230
MOVL C00231
MOVL C00232
MOVL C00233
MOVL C00234
MOVL C00235
MOVL C00236
MOVL C00237
MOVL C00238
MOVL C00239
MOVL C00240
MOVL C00241
MOVL C00242
MOVL C00243
MOVL C00244
MOVL C00245
MOVL C00246
MOVL C00247
MOVL C00248
MOVL C00249
MOVL C00250
MOVL C00251
MOVL C00252
MOVL C00253
MOVL C00254
MOVL C00255
MOVL C00256
MOVL C00257
MOVL C00258
MOVL C00259
MOVL C00260
MOVL C00261
MOVL C00262
MOVL C00263
MOVL C00264
MOVL C00265
MOVL C00266
MOVL C00267
MOVL C00268
MOVL C00269
MOVL C00270
MOVL C00271
MOVL C00272
MOVL C00273
MOVL C00274
MOVL C00275
MOVL C00276
MOVL C00277
MOVL C00278
MOVL C00279
MOVL C00280
MOVL C00281
MOVL C00282
MOVL C00283
MOVL C00284
MOVL C00285
MOVL C00286
MOVL C00287
MOVL C00288
MOVL C00289
MOVL C00290
MOVL C00291
MOVL C00292
MOVL C00293
MOVL C00294
MOVL C00295
MOVL C00296
MOVL C00297
MOVL C00298
MOVL C00299
MOVL C00300
MOVL C00301
MOVL C00302
MOVL C00303
MOVL C00304
MOVL C00305
MOVL C00306
MOVL C00307
MOVL C00308
MOVL C00309
MOVL C00310
MOVL C00311
MOVL C00312
MOVL C00313
MOVL C00314
MOVL C00315
MOVL C00316
MOVL C00317
MOVL C00318
MOVL C00319
MOVL C00320
MOVL C00321
MOVL C00322
MOVL C00323
MOVL C00324
MOVL C00325
MOVL C00326
MOVL C00327
MOVL C00328
MOVL C00329
MOVL C00330
MOVL C00331
MOVL C00332
MOVL C00333
MOVL C00334
MOVL C00335
MOVL C00336
MOVL C00337
MOVL C00338
MOVL C00339
MOVL C00340
MOVL C00341
MOVL C00342
MOVL C00343
MOVL C00344
MOVL C00345
MOVL C00346
MOVL C00347
MOVL C00348
MOVL C00349
MOVL C00350
MOVL C00351
MOVL C00352
MOVL C00353
MOVL C00354
MOVL C00355
MOVL C00356
MOVL C00357
MOVL C00358
MOVL C00359
MOVL C00360
MOVL C00361
MOVL C00362
MOVL C00363
MOVL C00364
MOVL C00365
MOVL C00366
MOVL C00367
MOVL C00368
MOVL C00369
MOVL C00370
MOVL C00371
MOVL C00372
MOVL C00373
MOVL C00374
MOVL C00375
MOVL C00376
MOVL C00377
MOVL C00378
MOVL C00379
MOVL C00380
MOVL C00381
MOVL C00382
MOVL C00383
MOVL C00384
MOVL C00385
MOVL C00386
MOVL C00387
MOVL C00388
MOVL C00389
MOVL C00390
MOVL C00391
MOVL C00392
MOVL C00393
MOVL C00394
MOVL C00395
MOVL C00396
MOVL C00397
MOVL C00398
MOVL C00399
MOVL C00400
MOVL C00401
MOVL C00402
MOVL C00403
MOVL C00404
MOVL C00405
MOVL C00406
MOVL C00407
MOVL C00408
MOVL C00409
MOVL C00410
MOVL C00411
MOVL C00412
MOVL C00413
MOVL C00414
MOVL C00415
MOVL C00416
MOVL C00417
MOVL C00418
MOVL C00419
MOVL C00420
MOVL C00421
MOVL C00422
MOVL C00423
MOVL C00424
MOVL C00425
MOVL C00426
MOVL C00427
MOVL C00428
MOVL C00429
MOVL C00430
MOVL C00431
MOVL C00432
MOVL C00433
MOVL C00434
MOVL C00435
MOVL C00436
MOVL C00437
MOVL C00438
MOVL C00439
MOVL C00440
MOVL C00441
MOVL C00442
MOVL C00443
MOVL C00444
MOVL C00445
MOVL C00446
MOVL C00447
MOVL C00448
MOVL C00449
MOVL C00450
MOVL C00451
MOVL C00452
MOVL C00453
MOVL C00454
ARCOF
MOVL C00455
ARCON
MOVL C00456
MOVL C00457
MOVL C00458
MOVL C00459
MOVL C00460
MOVL C00461
MOVL C00462
MOVL C00463
MOVL C00464
MOVL C00465
MOVL C00466
MOVL C00467
MOVL C00468
MOVL C00469
MOVL C00470
MOVL C00471
MOVL C00472
MOVL C00473
ARCOF
MOVL C00474
ARCON
MOVL C00475
MOVL C00476
MOVL C00477
MOVL C00478
MOVL C00479
MOVL C00480
MOVL C00481
MOVL C00482
MOVL C00483
MOVL C00484
MOVL C00485
MOVL C00486
MOVL C00487
MOVL C00488
MOVL C00489
MOVL C00490
MOVL C00491
MOVL C00492
ARCOF
MOVL C00493
ARCON
MOVL C00494
MOVL C00495
MOVL C00496
MOVL C00497
MOVL C00498
MOVL C00499
MOVL C00500
MOVL C00501
MOVL C00502
MOVL C00503
MOVL C00504
MOVL C00505
MOVL C00506
MOVL C00507
MOVL C00508
MOVL C00509
MOVL C00510
MOVL C00511
ARCOF
MOVL C00512
ARCON
MOVL C00513
MOVL C00514
MOVL C00515
MOVL C00516
MOVL C00517
MOVL C00518
MOVL C00519
MOVL C00520
MOVL C00521
MOVL C00522
MOVL C00523
MOVL C00524
MOVL C00525
MOVL C00526
MOVL C00527
MOVL C00528
MOVL C00529
MOVL C00530
MOVL C00531
ARCOF
MOVL C00532
ARCON
MOVL C00533
MOVL C00534
MOVL C00535
MOVL C00536
MOVL C00537
MOVL C00538
MOVL C00539
MOVL C00540
MOVL C00541
MOVL C00542
MOVL C00543
MOVL C00544
MOVL C00545
MOVL C00546
MOVL C00547
MOVL C00548
MOVL C00549
MOVL C00550
ARCOF
MOVL C00551
ARCON
MOVL C00552
MOVL C00553
MOVL C00554
MOVL C00555
MOVL C00556
MOVL C00557
MOVL C00558
MOVL C00559
MOVL C00560
MOVL C00561
MOVL C00562
MOVL C00563
MOVL C00564
MOVL C00565
MOVL C00566
MOVL C00567
MOVL C00568
MOVL C00569
ARCOF
MOVL C00570
ARCON
MOVL C00571
MOVL C00572
MOVL C00573
MOVL C00574
MOVL C00575
MOVL C00576
MOVL C00577
MOVL C00578
MOVL C00579
MOVL C00580
MOVL C00581
MOVL C00582
MOVL C00583
MOVL C00584
MOVL C00585
MOVL C00586
MOVL C00587
MOVL C00588
ARCOF
MOVL C00589
ARCON
MOVL C00590
MOVL C00591
MOVL C00592
MOVL C00593
MOVL C00594
MOVL C00595
MOVL C00596
MOVL C00597
MOVL C00598
MOVL C00599
MOVL C00600
MOVL C00601
MOVL C00602
MOVL C00603
MOVL C00604
ARCOF
MOVL C00605
ARCON
MOVL C00606
MOVL C00607
MOVL C00608
MOVL C00609
MOVL C00610
MOVL C00611
MOVL C00612
MOVL C00613
MOVL C00614
MOVL C00615
ARCOF
MOVL C00616
ARCON
MOVL C00617
MOVL C00618
MOVL C00619
MOVL C00620
MOVL C00621
MOVL C00622
MOVL C00623
MOVL C00624
MOVL C00625
MOVL C00626
ARCOF
MOVL C00627
ARCON
MOVL C00628
MOVL C00629
MOVL C00630
MOVL C00631
MOVL C00632
MOVL C00633
MOVL C00634
MOVL C00635
MOVL C00636
MOVL C00637
ARCOF
MOVL C00638
ARCON
MOVL C00639
MOVL C00640
MOVL C00641
MOVL C00642
MOVL C00643
MOVL C00644
MOVL C00645
MOVL C00646
MOVL C00647
MOVL C00648
MOVL C00649
ARCOF
MOVL C00650
ARCON
MOVL C00651
MOVL C00652
MOVL C00653
MOVL C00654
MOVL C00655
MOVL C00656
MOVL C00657
MOVL C00658
MOVL C00659
MOVL C00660
ARCOF
MOVL C00661
ARCON
MOVL C00662
MOVL C00663
MOVL C00664
MOVL C00665
MOVL C00666
MOVL C00667
MOVL C00668
MOVL C00669
MOVL C00670
MOVL C00671
ARCOF
MOVL C00672
ARCON
MOVL C00673
MOVL C00674
MOVL C00675
MOVL C00676
MOVL C00677
MOVL C00678
MOVL C00679
MOVL C00680
MOVL C00681
MOVL C00682
ARCOF
MOVL C00683
ARCON
MOVL C00684
MOVL C00685
MOVL C00686
MOVL C00687
MOVL C00688
MOVL C00689
MOVL C00690
MOVL C00691
MOVL C00692
MOVL C00693
ARCOF
MOVL C00694
ARCON
MOVL C00695
MOVL C00696
MOVL C00697
MOVL C00698
MOVL C00699
MOVL C00700
MOVL C00701
MOVL C00702
ARCOF
MOVL C00703
ARCON
MOVL C00704
MOVL C00705
MOVL C00706
MOVL C00707
MOVL C00708
MOVL C00709
MOVL C00710
MOVL C00711
ARCOF
MOVL C00712
ARCON
MOVL C00713
MOVL C00714
MOVL C00715
MOVL C00716
MOVL C00717
MOVL C00718
MOVL C00719
MOVL C00720
ARCOF
MOVL C00721
ARCON
MOVL C00722
MOVL C00723
MOVL C00724
MOVL C00725
MOVL C00726
MOVL C00727
MOVL C00728
MOVL C00729
MOVL C00730
ARCOF
MOVL C00731
ARCON
MOVL C00732
MOVL C00733
MOVL C00734
MOVL C00735
MOVL C00736
MOVL C00737
MOVL C00738
MOVL C00739
ARCOF
MOVL C00740
ARCON
MOVL C00741
MOVL C00742
MOVL C00743
MOVL C00744
MOVL C00745
MOVL C00746
MOVL C00747
MOVL C00748
ARCOF
MOVL C00749
ARCON
MOVL C00750
MOVL C00751
MOVL C00752
MOVL C00753
MOVL C00754
MOVL C00755
MOVL C00756
MOVL C00757
ARCOF
MOVL C00758
ARCON
MOVL C00759
MOVL C00760
MOVL C00761
MOVL C00762
MOVL C00763
MOVL C00764
MOVL C00765
MOVL C00766
ARCOF
MOVL C00767
ARCON
MOVL C00768
MOVL C00769
MOVL C00770
MOVL C00771
MOVL C00772
MOVL C00773
ARCOF
MOVL C00774
ARCON
MOVL C00775
MOVL C00776
MOVL C00777
MOVL C00778
MOVL C00779
MOVL C00780
ARCOF
MOVL C00781
ARCON
MOVL C00782
MOVL C00783
MOVL C00784
MOVL C00785
MOVL C00786
MOVL C00787
ARCOF
MOVL C00788
ARCON
MOVL C00789
MOVL C00790
MOVL C00791
MOVL C00792
MOVL C00793
MOVL C00794
MOVL C00795
ARCOF
MOVL C00796
ARCON
MOVL C00797
MOVL C00798
MOVL C00799
MOVL C00800
MOVL C00801
MOVL C00802
ARCOF
MOVL C00803
ARCON
MOVL C00804
MOVL C00805
MOVL C00806
MOVL C00807
MOVL C00808
MOVL C00809
ARCOF
MOVL C00810
ARCON
MOVL C00811
MOVL C00812
MOVL C00813
MOVL C00814
MOVL C00815
MOVL C00816
ARCOF
MOVL C00817
ARCON
MOVL C00818
MOVL C00819
MOVL C00820
END
